// TIA Portal project "ısı_basınç_kontrol" (V18)

(* hardware
DEVICE "S7-1200 station_1"  S7-1200 Station
   slot 0: "Rack_0"  S7-1200 Rack  Rack  V1.0
   slot 1: "PLC_1"  CPU 1212C DC/DC/DC  6ES7 212-1AE40-0XB0  V4.6
*)

// ===== PLC "PLC_1"  CPU 1212C DC/DC/DC =====

VAR_GLOBAL   // PLC tag table "Default tag table"
   "high_pressure" AT %I0.0 : Bool;
   "low_pressure" AT %I0.1 : Bool;
   "high_temp" AT %I0.2 : Bool;
   "low_temp" AT %I0.3 : Bool;
   "mixer" AT %Q0.0 : Bool;
   "relief valve" AT %Q0.1 : Bool;
   "cold_water_inlet" AT %Q0.2 : Bool;
   "heater" AT %Q0.3 : Bool;
   "start" AT %Q0.4 : Bool;
   "normal_operation" AT %Q0.5 : Bool;
   "alarm" AT %Q0.6 : Bool;
END_VAR

FUNCTION "Block_1" : Void   // FC1, LAD
{ S7_Optimized_Access := 'TRUE' }
VERSION : 0.1
BEGIN

REGION Network 1
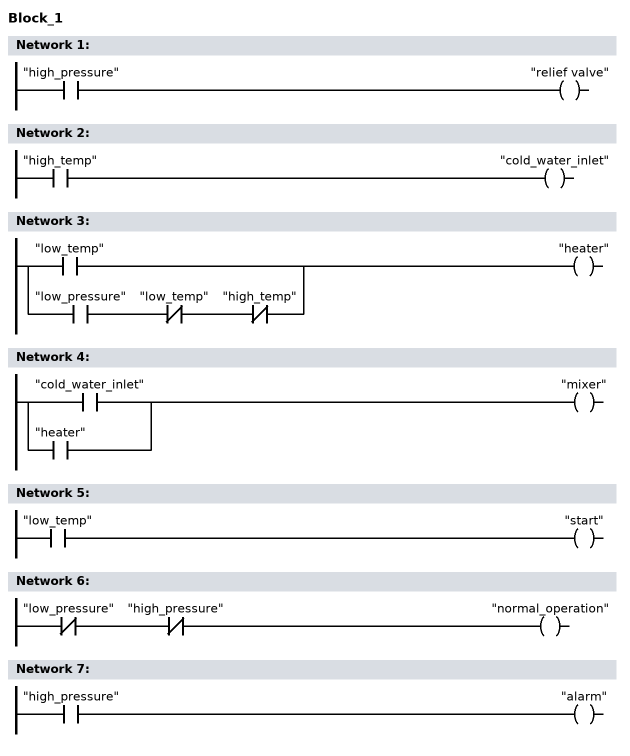
   RUNG wire#powerrail
      Contact( "high_pressure" )
      Coil( "relief valve" )
   END_RUNG
   // the same network as SCL:
   "relief valve" := "high_pressure";
END_REGION

REGION Network 2
   RUNG wire#powerrail
      Contact( "high_temp" )
      Coil( "cold_water_inlet" )
   END_RUNG
   // the same network as SCL:
   "cold_water_inlet" := "high_temp";
END_REGION

REGION Network 3
   RUNG wire#powerrail
      Contact( "low_temp" )
      wire#w1
      Coil( "heater" )
   END_RUNG
   RUNG wire#powerrail
      Contact( "low_pressure" )
      I_Contact( "low_temp" )
      I_Contact( "high_temp" )
   END_RUNG wire#w1
   // the same network as SCL:
   "heater" := "low_temp" OR ("low_pressure" AND NOT "low_temp" AND NOT "high_temp");
END_REGION

REGION Network 4
   RUNG wire#powerrail
      Contact( "cold_water_inlet" )
      wire#w1
      Coil( "mixer" )
   END_RUNG
   RUNG wire#powerrail
      Contact( "heater" )
   END_RUNG wire#w1
   // the same network as SCL:
   "mixer" := "cold_water_inlet" OR "heater";
END_REGION

REGION Network 5
   RUNG wire#powerrail
      Contact( "low_temp" )
      Coil( "start" )
   END_RUNG
   // the same network as SCL:
   "start" := "low_temp";
END_REGION

REGION Network 6
   RUNG wire#powerrail
      I_Contact( "low_pressure" )
      I_Contact( "high_pressure" )
      Coil( "normal_operation" )
   END_RUNG
   // the same network as SCL:
   "normal_operation" := NOT "low_pressure" AND NOT "high_pressure";
END_REGION

REGION Network 7
   RUNG wire#powerrail
      Contact( "high_pressure" )
      Coil( "alarm" )
   END_RUNG
   // the same network as SCL:
   "alarm" := "high_pressure";
END_REGION
END_FUNCTION

ORGANIZATION_BLOCK "Main"   // OB1, LAD, ProgramCycle
TITLE = "Main Program Sweep (Cycle)"
{ S7_Optimized_Access := 'TRUE' }
VERSION : 0.1
   VAR_INPUT
      Initial_Call : Bool;   // Initial call of this OB
      Remanence : Bool;   // =True, if remanent data are available
   END_VAR
BEGIN

REGION Network 1
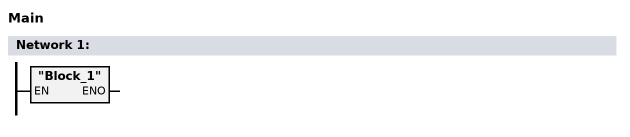
   RUNG wire#powerrail
      "Block_1"()
   END_RUNG
   // the same network as SCL:
   "Block_1"();
END_REGION
END_ORGANIZATION_BLOCK